//==================================================================================================
//							Beckhoff Automation Poland
//								FB_AntiBlinkAlarmFilter
//									20.12.2016
//				Blok służący do wyłączania logowania zdarzeń które pojawiają się zbyt często
// 	v1.0 || TC v 3.1.4020.28 || - pierwsza wersja
//==================================================================================================
FUNCTION_BLOCK FB_AntiBlinkAlarmFilter
VAR_INPUT
	bEvent			: BOOL;		// Status zdarzenia
	tTime			: TIME;		// Zadane okno czasowe
	uiLimit			: UINT;		// Maksymalna liczba zdarzeń jaka może się pojawić w oknie czasowym
END_VAR
VAR_IN_OUT
	bPermission		: BOOL;		// Flaga zezwolenia na logowanie zdarzeń
END_VAR
VAR
	tStartTime		: TIME;		// Zmienna przechowująca czas rozpoczęcia zliczania
	uiActCount		: UINT;		// Aktualna wartość licznika
	rtEdge			: R_TRIG;	// Zbocze narastające
END_VAR

rtEdge(CLK:=bEvent);
IF rtEdge.Q THEN							// Blok podejmuje akcję w przypadku wystapienia zdarzenia
	IF uiActCount = 0 THEN	
		tStartTime		:= TIME();			// W przypadku gdy licznik wynosi zero, zapisywany jest czas rozpoczęcia zliczania
	END_IF
	uiActCount			:= uiActCount + 1;	// Inkrementacja licznika liczby zdarzeń
	IF uiActcount >= uiLimit THEN			// W przypadku gdy liczba zdarzeń osiągnie zadany limit, sprawdzany jest czas w jakim one wystapiły. Jeśli czas jest większy niż dopuszczalny, resetowana jest flaga zezwolenia
		IF TIME() - tStartTime < tTime THEN
			bPermission	:= FALSE;		
		END_IF
		uiActCount 		:= 0;
	END_IF
	IF NOT bPermission THEN
		uiActCount		:= 0;
	END_IF
END_IF;

END_FUNCTION_BLOCK

(* stored: Version 1.1.0.1, ProductVersion 3.1.4026.13, FileIdentifier 578989723503ad64b5723de191a4159a5d91c67b, FileSignature 43eb0d6f867ed4cdffb9f135d01a764f6a1d6ef86c9fad24cb10e21d2a91fbaf33d15d2209f1484a5f1b5048e1e7ffbea724bcc021f4aed852222781cbec6fe29fd7d900f2c627cd9aff8ff934c2b944dddd77b9c3bc80c06351e8b4fdb4fe1c1e4632265a4b67ca0f6e92a999e9bd95582652f2ced22792d0b956265192d6a2d71b22af1f2ef69f2e05f6fe1329ab1a2240e6b0487ec11cab923c452ca600ffceca113b687456bc7073e33b778407b6b29437659a2588f0362ae28962c6ccce5f7308d823ea1575cbce4fd60c9a7f527ac341c6ad798a0c71702c739f2a34ca29e47825d55645dceeff4803258fe37a110f16b347ebd017b12479e1830bf6a9
   POU FB_AntiBlinkAlarmFilter: Id {ee86e843-ab76-4901-a36e-d9e2f7a1a2fa}, SpecialFunc None *)
